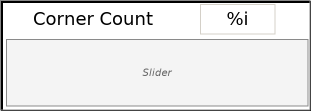
VISUALIZATION InputNumSlider_Corner  // 311x111
    Rectangle (1,1 310x110)
    Label (30,4 150x30), "Corner Count"
    Textfield (200,4 75x30), "%i", text variable: MAIN.FB_FigureGenerator.nCornerCountInp
        OnMouseClick: write the text variable via Default, min 3, max 100
    Slider (6,39 302x67), variable: MAIN.FB_FigureGenerator.nCornerCountInp, scale 3..13
END_VISUALIZATION

(* stored: Version 1.1.0.1, ProductVersion 3.1.4024.12
   Visu InputNumSlider_Corner: Id {96a97254-8599-42e3-bfab-09ee7a10b194} *)
